Omron CX-Programmer project NewProject (CX-Programmer 9.51)

# PLC my_first_project: CP1L L
; Comment

## Program NewProgram1 (cyclic task 0)
Local symbols
button_1 0.00 BOOL  ; Comment
button_2 0.01 BOOL  ; Comment
buttton_3 0.02 BOOL
out_2 100.01 BOOL  ; Comment
out_3 100.02 BOOL  ; Commment

### Section Section1

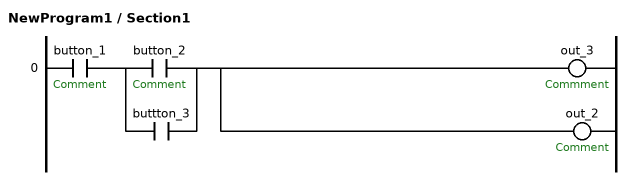
; rung 0
LD button_1  ; Comment
LD button_2  ; Comment
OR buttton_3
ANDLD
OUT out_3  ; Commment
OUT out_2  ; Comment

### Section END
; rung 0
END(001)